(* Passes one UDINT read across the arbiter bridge. The caller links the raw PDO value and derives
   bridge health elsewhere (e.g. FB_SubSysToArbiter_IO.bBridgeOk) and passes both in each cycle; this
   FB owns no hardware links. Integers have no invalid-bit-pattern to sanitize, so it holds the last
   trusted value while the bridge is down. Error carries only the test override; fault on bad comms
   via the bridge FB's bBridgeConfirmedBad in the caller. *)
FUNCTION_BLOCK FB_FallibleUdintFromEtherCAT
IMPLEMENTS I_FallibleUdint
VAR_INPUT
    i_bBridgeOk : BOOL;
    i_nValue : UDINT;
END_VAR
VAR_OUTPUT
    {attribute 'pytmc' := '
        pv: Value
        io: i
    '}
    nValue : UDINT;
END_VAR
VAR
    nLastValidValue : UDINT;
    bOverride : BOOL;
    bOverrideError : BOOL;
    nOverrideValue : UDINT;
END_VAR


IF i_bBridgeOk THEN
    nLastValidValue := i_nValue;
END_IF

nValue := SEL(bOverride, SEL(i_bBridgeOk, nLastValidValue, i_nValue), nOverrideValue);


PROPERTY Error : BOOL
GET

Error := SEL(bOverride, FALSE, bOverrideError);
END_GET
END_PROPERTY


PROPERTY Value : UDINT
GET

Value := THIS^.nValue;
END_GET
END_PROPERTY

END_FUNCTION_BLOCK

(* stored: Version 1.1.0.1
   POU FB_FallibleUdintFromEtherCAT: Id {a1b2c3d4-0103-4001-8001-000000000301}, SpecialFunc None
   Property Error: Id {a1b2c3d4-0103-4001-8001-000000000302}
   Get Get: Id {a1b2c3d4-0103-4001-8001-000000000303}
   Property Value: Id {a1b2c3d4-0103-4001-8001-000000000304}
   Get Get: Id {a1b2c3d4-0103-4001-8001-000000000305} *)
